FUNCTION "FC_SimRedler" : Void
{ S7_Optimized_Access := 'TRUE' }
VERSION : 2.1
// ==============================================================================
// FC_SimRedler - Симулятор фізики та несправностей редлера
// ==============================================================================
// Версія: 2.1.0
// Дата: 2026-04-10
// ==============================================================================
// Зміни v2.1:
//   + Додано симуляцію DI_Speed_OK (PHASE 2) — тахо
//   + Додано симуляцію SimFault_Breaker та SimFault_Overflow
// ==============================================================================
// Комунікація з FC_Redler ТІЛЬКИ через сигнали:
//   - Читає:  DB_Mechs.Redler[RedlerIdx].DO_Run
//   - Пише:   DB_Mechs.Redler[RedlerIdx].DI_Speed_OK
//             DB_Mechs.Redler[RedlerIdx].DI_Breaker_OK
//             DB_Mechs.Redler[RedlerIdx].DI_Overflow_OK
// ==============================================================================
   VAR_INPUT
      RedlerIdx : Int;
      StartupTime_ms : DInt;
      StopTime_ms : DInt;
      SimFault_Breaker : Bool;
      FaultTime_Breaker_ms : DInt;
      SimFault_Overflow : Bool;
      FaultTime_Overflow_ms : DInt;
      ManualReset : Bool;
   END_VAR

   VAR_TEMP
      idx : Int;
      elapsedMs : DInt;
      nowTck : DInt;
      startupTimeout : Bool;
      stopTimeout : Bool;
      breakerTimeout : Bool;
      overflowTimeout : Bool;
   END_VAR


BEGIN
	    // =========================================================
	    // VALIDATE INDEX
	    // =========================================================
	    IF #RedlerIdx >= "REDLERS_COUNT"+1 THEN
	        RETURN;
	    END_IF;

	    #idx := #RedlerIdx;

	    // =========================================================
	    // PHASE 0: Ручний скид аварій
	    // =========================================================
	    IF #ManualReset THEN
	        "DB_SimMechs".Redler[#idx].Breaker_Tripped := FALSE;
	        "DB_SimMechs".Redler[#idx].Overflow_Tripped := FALSE;
	END_IF;
	    IF "DB_Mechs".Redler[#idx].DO_Run AND NOT "DB_SimMechs".Redler[#idx].LastDO_Run THEN
	        "DB_SimMechs".Redler[#idx].MotorStartTck := TIME_TCK();
	        "DB_SimMechs".Redler[#idx].FaultStartTck := TIME_TCK();
	        "DB_SimMechs".Redler[#idx].IsMotorRunning := TRUE;
	        "DB_SimMechs".Redler[#idx].IsSpinningUp := TRUE;
	        "DB_SimMechs".Redler[#idx].IsSpinningDown := FALSE;
	    END_IF;

	    IF NOT "DB_Mechs".Redler[#idx].DO_Run AND "DB_SimMechs".Redler[#idx].LastDO_Run THEN
	        "DB_SimMechs".Redler[#idx].MotorStopTck := TIME_TCK();
	        "DB_SimMechs".Redler[#idx].IsMotorRunning := FALSE;
	        "DB_SimMechs".Redler[#idx].IsSpinningUp := FALSE;
	        "DB_SimMechs".Redler[#idx].IsSpinningDown := TRUE;
	    END_IF;

	    "DB_SimMechs".Redler[#idx].LastDO_Run := "DB_Mechs".Redler[#idx].DO_Run;

	    // =========================================================
	    // PHASE 2: Симуляція DI_Speed_OK (тахо)
	    // =========================================================
	    IF "DB_SimMechs".Redler[#idx].IsSpinningUp THEN
	        #startupTimeout := "FC_TimeElapsedMs"(
	                                              StartTck := "DB_SimMechs".Redler[#idx].MotorStartTck,
	                                              TimeoutMs := #StartupTime_ms,
	                                              ElapsedMs => #elapsedMs,
	                                              NowTck => #nowTck
	        );
	        IF #startupTimeout THEN
	            "DB_Mechs".Redler[#idx].DI_Speed_OK := TRUE;
	            "DB_SimMechs".Redler[#idx].IsSpinningUp := FALSE;
	        ELSE
	            "DB_Mechs".Redler[#idx].DI_Speed_OK := FALSE;
	        END_IF;
	    ELSIF "DB_SimMechs".Redler[#idx].IsSpinningDown THEN
	        #stopTimeout := "FC_TimeElapsedMs"(
	                                           StartTck := "DB_SimMechs".Redler[#idx].MotorStopTck,
	                                           TimeoutMs := #StopTime_ms,
	                                           ElapsedMs => #elapsedMs,
	                                           NowTck => #nowTck
	        );
	        IF #stopTimeout THEN
	            "DB_Mechs".Redler[#idx].DI_Speed_OK := FALSE;
	            "DB_SimMechs".Redler[#idx].IsSpinningDown := FALSE;
	        ELSE
	            "DB_Mechs".Redler[#idx].DI_Speed_OK := TRUE;
	        END_IF;
	    ELSIF "DB_SimMechs".Redler[#idx].IsMotorRunning THEN
	        "DB_Mechs".Redler[#idx].DI_Speed_OK := TRUE;
	    ELSE
	        "DB_Mechs".Redler[#idx].DI_Speed_OK := FALSE;
	    END_IF;

	    // =========================================================
	    // PHASE 4: Симуляція аварії BREAKER
	    // =========================================================
	    IF #SimFault_Breaker AND "DB_SimMechs".Redler[#idx].IsMotorRunning AND NOT "DB_SimMechs".Redler[#idx].Breaker_Tripped THEN
	        #breakerTimeout := "FC_TimeElapsedMs"(
	                                              StartTck := "DB_SimMechs".Redler[#idx].FaultStartTck,
	                                              TimeoutMs := #FaultTime_Breaker_ms,
	                                              ElapsedMs => #elapsedMs,
	                                              NowTck => #nowTck
	        );
	        IF #breakerTimeout THEN
	            "DB_SimMechs".Redler[#idx].Breaker_Tripped := TRUE;
	        END_IF;
	    END_IF;
	    "DB_Mechs".Redler[#idx].DI_Breaker_OK := NOT "DB_SimMechs".Redler[#idx].Breaker_Tripped;

	    // =========================================================
	    // PHASE 5: Симуляція аварії OVERFLOW
	    // =========================================================
	    IF #SimFault_Overflow AND "DB_SimMechs".Redler[#idx].IsMotorRunning AND NOT "DB_SimMechs".Redler[#idx].Overflow_Tripped THEN
	        #overflowTimeout := "FC_TimeElapsedMs"(
	                                               StartTck := "DB_SimMechs".Redler[#idx].FaultStartTck,
	                                               TimeoutMs := #FaultTime_Overflow_ms,
	                                               ElapsedMs => #elapsedMs,
	                                               NowTck => #nowTck
	        );
	        IF #overflowTimeout THEN
	            "DB_SimMechs".Redler[#idx].Overflow_Tripped := TRUE;
	        END_IF;
	    END_IF;
	    "DB_Mechs".Redler[#idx].DI_Overflow_OK := NOT "DB_SimMechs".Redler[#idx].Overflow_Tripped;

	    // =========================================================

END_FUNCTION
